TYPE sRoboterProzessVariablen :
STRUCT
	q1					:LREAL;				// X-Koordinate oder Gelenkwinkel 1
	q2					:LREAL;				// Y-Koordinate oder Gelenkwinkel 2
	q3					:LREAL;				// Z-Koordinate oder Gelenkwinkel 3
	q4					:LREAL;				// Orintierung um X-Achse oder Gelenkwinkel 4
	q5					:LREAL;				// Orientierung um Y-Achse oder Gelenkwinkel 5
	q6					:LREAL;				// Orientierung um Z-Achse oder Gelenkwinkel 6
	v					:LREAL;				// Geschwindigkeit
	a					:LREAL;				// Beschleunigung
	PosTyp				:eRobPosType;		// Position-Typ definieren (Absolut / Relativ)		
	MoveTyp				:eRobMoveType;		// Bewegungsart definieren (Linear / Circular etc.)
END_STRUCT
END_TYPE

(* stored: Version 1.1.0.1
   DUT sRoboterProzessVariablen: Id {33686f70-1b98-41fe-b1f3-24a9ebb5410a} *)
